FUNCTION_BLOCK Test_DateTimeAsString EXTENDS TUnitTestBase
VAR
END_VAR

METHOD  Execute
VAR_INST
    TimeStruct : TIMESTRUCT := (wDay := 23, wMonth := 12, wYear := 1945, wHour := 22, wMinute := 20, wSecond := 18);
END_VAR
Assertion.AssertEquals_STRING(
    Expected := '22:20:18 23/12/1945',
    Actual   := F_DateTimeAsString(TimeStruct),
    ObjectName := _TestName,
    VariableName  := 'F_DateTimeAsString(TimeStruct)');


Test_Finished();
END_METHOD

END_FUNCTION_BLOCK

(* stored: Version 1.1.0.1, ProductVersion 3.1.4024.3
   POU Test_DateTimeAsString: Id {aa9aead4-27c1-4eae-ab82-d0277f89d638}, SpecialFunc None
   Method Execute: Id {1b97fda2-2485-425c-8310-a5715d5a1f54} *)
